VAR_GLOBAL
	dtVariable : DATE_AND_TIME := DT#2023-02-08-15:31:19;
	pToString : POINTER TO STRING;
	var2 : TIME := T#5S;
	var2Ref: REFERENCE TO TIME;
	var3 : ARRAY[1..4] OF DATE := [D#2023-02-7, D#2023-02-8, D#2023-02-9, D#2023-02-10];
	
	Sensor1 : Sensies := Sensies.Parker;
	
	TimeToPass : TIME := T#10S;
	Timmie : TON := (PT := TimeToPass);
	StartTimer : BOOL := FALSE;
	CurrentTimmie : TIME;
	IsFinished : BOOL;
	
END_VAR

(* stored: Version 1.1.0.1, ProductVersion 3.1.4024.12
   GVL DB: Id {cfcd30fd-6e5e-4ca5-9db1-0ada0c0c00a7} *)
